Universal Robots PolyScope program: Coexistence_PickAndPlace.urp

Program Coexistence_PickAndPlace (installation=Coexistence_PickAndPlace directory=/home/cobot/ursim-5.11.5.1010327/programs createdIn=5.11.5.1010327 lastSavedIn=5.11.5.1010327 robotSerialNumber=20195599999)
Calibrated DH parameters: a=[0, -0.425, -0.3922, 0, 0, 0]; d=[0.1625, 0, 0, 0.1333, 0.0997, 0.0996]; alpha=[1.570796, 0, 0, 1.570796, -1.570796, 0]; deltaTheta=[0, 0, 0, 0, 0, 0]
Robot Program (runOnlyOnce=false)
  Wait DigitalInput pin=GP_bool_in[64]; digitalValue=1
  Switch expression=GP_int_in[24]
    Case (caseValue=1)
      'Move to Home position'
      SafeHome (positionOptionType=SPEED_AND_ACCELERATION speed=1.047198 acceleration=1.396263 nextMotionTime=2)
    Case (caseValue=2)
      'Read new position and active workspace and move there'
      Pos := p[GP_float_in[24],GP_float_in[25],GP_float_in[26],GP_float_in[27],GP_float_in[28],GP_float_in[29]]
      Switch expression=GP_int_in[25]
        Case (caseValue=0)
          MoveJ speed 60 deg/s, acceleration 80 deg/s^2 (useActiveTCP=true) feature=Partbox
            Waypoint Waypoint (Variable): variable=Pos
        Case (caseValue=1)
          MoveJ speed 60 deg/s, acceleration 80 deg/s^2 (useActiveTCP=true) feature=Placelocation
            Waypoint Waypoint (Variable): variable=Pos
    Case (caseValue=3)
      'Pick part (simulated by wait)'
      Wait Sleep waitTime=2
    Case (caseValue=4)
      'Lift part (lift 20cm)'
      MoveL speed 250 mm/s, acceleration 1200 mm/s^2 (useActiveTCP=true) feature=Partbox
        MoveDirectionNode (selectedDirection=ZPlus)
          Until DISTANCE (allowActions=false deceleration=3 distanceNodeType=STOP) Distance=0.2; motionParameters(blendRadius=0)
    Case (caseValue=5)
      'Place part (simulated by wait)'
      Wait Sleep waitTime=2
      MoveL speed 250 mm/s, acceleration 1200 mm/s^2 (useActiveTCP=true) feature=Placelocation
        MoveDirectionNode (selectedDirection=ZPlus)
          Until DISTANCE (allowActions=false deceleration=3 distanceNodeType=STOP) Distance=0.1; motionParameters(blendRadius=0)
    Case (caseValue=2147483647)
      'Do nothing (just handshake)'
  Set DigitalOutput pin=GP_bool_out[64]; digitalValue=1
  Wait DigitalInput pin=GP_bool_in[64]; digitalValue=0
  Set DigitalOutput pin=GP_bool_out[64]; digitalValue=0
